PROGRAM PRG_TEST
VAR
	FB_Beckhoff_EL5002_Test : FB_Beckhoff_EL5002_Test;
END_VAR

TcUnit.RUN();

END_PROGRAM

(* stored: Version 1.1.0.1, ProductVersion 3.1.4024.12
   POU PRG_TEST: Id {bd0cd056-c9be-07e2-1020-9a5696ebe527}, SpecialFunc None *)
